(* Logix 5000 project; controller SolisPLC_CLX1 vendor 1 type 14 code 54 rev 20.19; software revision 20.04 *)

TASK MainTask (continuous, watchdog 500 ms) : MainProgram

MODULES
   Local : vendor 1 type 14 code 54 (ICP 0, rev 20.19)
      EN2T : 1756-EN2T (ICP 1, Ethernet 192.168.1.30, rev 5.1, Input RPI 500 ms)
         Kinetix350_MTR1 : vendor 1 type 37 code 32 (Ethernet 192.168.1.14, rev 2.1, MotionDiagnostics RPI 1 ms, MotionSync RPI 1 ms)
END_MODULES

VAR_GLOBAL   (* controller tags *)
   Axis1 : AXIS_CIP_DRIVE;
   Motion_G1 : MOTION_GROUP;
END_VAR

PROGRAM MainProgram   (* main routine MainRoutine *)

ROUTINE MainRoutine   (* ladder *)
END_ROUTINE
END_PROGRAM
